ABB RAPID module: tester_left.mod

MODULE tester_left
LOCAL CONST string YuMi_App_Program_Version:="1.0.1"; !Do not edit or remove this line!
LOCAL VAR robtarget p35 := [[358.29,68.3,132.84],[0.2751,-0.0426083,0.86319,-0.421199],[-1,1,0,11],[117.327,9E+09,9E+09,9E+09,9E+09,9E+09]];
LOCAL VAR robtarget p34 := [[519.08,52.62,111.62],[0.0190745,-0.317014,0.947041,-0.0474542],[-2,1,-2,11],[179.331,9E+09,9E+09,9E+09,9E+09,9E+09]];
LOCAL VAR robtarget p33 := [[488.88,196.13,-9.51],[0.0436672,0.774832,-0.594672,-0.209984],[-2,0,-2,11],[-128.122,9E+09,9E+09,9E+09,9E+09,9E+09]];
LOCAL VAR robtarget p32 := [[438.93,-11.04,-14.27],[0.137086,0.640295,-0.744056,-0.132704],[-2,0,-2,11],[-135.659,9E+09,9E+09,9E+09,9E+09,9E+09]];
LOCAL VAR robtarget p31 := [[346.07,2.52,-21.9],[0.183409,0.628509,-0.722146,-0.223252],[-2,0,-2,11],[-129.96,9E+09,9E+09,9E+09,9E+09,9E+09]];
LOCAL VAR robtarget p30 := [[346.36,2.76,-22.07],[0.182499,0.628074,-0.72283,-0.223011],[-2,0,-2,11],[-129.954,9E+09,9E+09,9E+09,9E+09,9E+09]];
LOCAL VAR robtarget p29 := [[346.36,2.76,-22.07],[0.182498,0.628074,-0.722831,-0.22301],[-2,0,-2,11],[-129.954,9E+09,9E+09,9E+09,9E+09,9E+09]];
LOCAL VAR robtarget p28 := [[346.36,2.76,-22.07],[0.182497,0.628073,-0.722832,-0.223009],[-2,0,-2,11],[-129.954,9E+09,9E+09,9E+09,9E+09,9E+09]];
LOCAL VAR robtarget p27 := [[346.36,2.76,-22.07],[0.182493,0.628073,-0.722833,-0.22301],[-2,0,-2,11],[-129.954,9E+09,9E+09,9E+09,9E+09,9E+09]];
LOCAL VAR robtarget p26 := [[346.36,2.76,-22.07],[0.182492,0.628071,-0.722834,-0.223011],[-2,0,-2,11],[-129.954,9E+09,9E+09,9E+09,9E+09,9E+09]];
LOCAL VAR robtarget p25 := [[346.36,2.76,-22.07],[0.182489,0.628071,-0.722835,-0.22301],[-2,0,-2,11],[-129.954,9E+09,9E+09,9E+09,9E+09,9E+09]];
LOCAL VAR robtarget p24 := [[346.37,2.77,-22.07],[0.182481,0.628066,-0.722841,-0.223011],[-2,0,-2,11],[-129.954,9E+09,9E+09,9E+09,9E+09,9E+09]];
LOCAL VAR robtarget p23 := [[346.37,2.77,-22.08],[0.182475,0.628061,-0.722847,-0.22301],[-2,0,-2,11],[-129.954,9E+09,9E+09,9E+09,9E+09,9E+09]];
LOCAL VAR robtarget p22 := [[346.37,2.77,-22.08],[0.182471,0.628058,-0.722852,-0.223008],[-2,0,-2,11],[-129.954,9E+09,9E+09,9E+09,9E+09,9E+09]];
LOCAL VAR robtarget p21 := [[346.37,2.77,-22.08],[0.182457,0.628053,-0.72286,-0.223006],[-2,0,-2,11],[-129.954,9E+09,9E+09,9E+09,9E+09,9E+09]];
LOCAL VAR robtarget p20 := [[346.39,2.81,-22.09],[0.182382,0.628009,-0.722913,-0.223019],[-2,0,-2,11],[-129.952,9E+09,9E+09,9E+09,9E+09,9E+09]];
LOCAL VAR robtarget p19 := [[346.92,3.05,-22.39],[0.18104,0.627419,-0.724003,-0.222238],[-2,0,-2,11],[-129.95,9E+09,9E+09,9E+09,9E+09,9E+09]];
LOCAL VAR robtarget p18 := [[367.84,3.92,14.47],[0.223286,0.640903,-0.702206,-0.215161],[-2,0,-2,11],[-130.827,9E+09,9E+09,9E+09,9E+09,9E+09]];
LOCAL VAR robtarget p17 := [[412.3,51.52,46.99],[0.26981,0.654674,-0.703812,-0.0570357],[-2,0,-2,11],[-126.803,9E+09,9E+09,9E+09,9E+09,9E+09]];
LOCAL VAR robtarget p16 := [[496.94,50.54,-0.5],[0.0852698,-0.611194,0.718186,-0.321526],[-2,0,-1,1010],[-139.426,9E+09,9E+09,9E+09,9E+09,9E+09]];
LOCAL VAR robtarget p15 := [[500.11,217.09,68.79],[0.372259,-0.540285,0.603529,-0.453064],[-2,0,-1,1010],[-136.231,9E+09,9E+09,9E+09,9E+09,9E+09]];
LOCAL VAR robtarget p14 := [[409.25,103.49,24.74],[0.422813,-0.52314,0.597648,-0.436314],[-2,0,-1,1010],[-146.03,9E+09,9E+09,9E+09,9E+09,9E+09]];
LOCAL VAR robtarget p13 := [[321.14,2.68,-3.7],[0.326511,-0.570175,0.616333,-0.434079],[-2,0,-1,1010],[-149.503,9E+09,9E+09,9E+09,9E+09,9E+09]];
LOCAL VAR robtarget p12 := [[323.71,20.37,-12.88],[0.347699,-0.567053,0.614733,-0.423862],[-2,0,-1,1010],[-149.327,9E+09,9E+09,9E+09,9E+09,9E+09]];
LOCAL VAR robtarget p11 := [[318.83,3.47,-66.12],[0.377646,-0.544178,0.635778,-0.396283],[-2,0,-1,1010],[-148.179,9E+09,9E+09,9E+09,9E+09,9E+09]];
LOCAL VAR robtarget p10 := [[319.84,5.22,-58.84],[0.383222,-0.546134,0.616372,-0.418288],[-2,0,-1,1010],[-147.982,9E+09,9E+09,9E+09,9E+09,9E+09]];
LOCAL VAR robtarget p9 := [[328.17,3.84,-35.32],[0.291971,-0.584613,0.689413,-0.312553],[-2,0,-1,1010],[-148.669,9E+09,9E+09,9E+09,9E+09,9E+09]];
LOCAL VAR robtarget p8 := [[337.64,30.76,-7.64],[0.0603166,-0.700953,0.706625,-0.0755479],[-2,-1,-1,1010],[-140.725,9E+09,9E+09,9E+09,9E+09,9E+09]];
LOCAL VAR robtarget p7 := [[339.22,39.97,2.31],[0.254333,0.704549,-0.624556,-0.221031],[-2,-2,0,1010],[-142.847,9E+09,9E+09,9E+09,9E+09,9E+09]];
LOCAL VAR robtarget p6 := [[280.93,-22.19,-89.26],[0.280661,0.753652,-0.552241,-0.219698],[-2,-2,0,1010],[-144.058,9E+09,9E+09,9E+09,9E+09,9E+09]];
LOCAL VAR robtarget p5 := [[282.32,-20.83,-89.42],[0.275747,0.742915,-0.569862,-0.217482],[-2,-2,0,1010],[-144.216,9E+09,9E+09,9E+09,9E+09,9E+09]];
LOCAL VAR robtarget p4 := [[286.48,-20.76,-86.12],[0.126721,0.794038,-0.590704,-0.0671829],[-2,-1,-1,1010],[-143.981,9E+09,9E+09,9E+09,9E+09,9E+09]];
LOCAL VAR robtarget p3 := [[304.13,-11.5,-50.26],[0.0519145,0.826957,-0.559517,-0.0197134],[-2,-1,-1,1010],[-154.754,9E+09,9E+09,9E+09,9E+09,9E+09]];
LOCAL VAR robtarget p2 := [[316.65,45.52,21.47],[0.0502929,0.702983,-0.635561,0.315196],[-1,0,-1,1010],[-169.577,9E+09,9E+09,9E+09,9E+09,9E+09]];
LOCAL VAR robtarget p1 := [[358.29,68.3,132.84],[0.275101,-0.0426095,0.86319,-0.421198],[-1,1,0,11],[117.327,9E+09,9E+09,9E+09,9E+09,9E+09]];
LOCAL VAR robtarget s35 := [[358.29,68.3,132.84],[0.2751,-0.0426083,0.86319,-0.421199],[-1,1,0,11],[117.327,9E+09,9E+09,9E+09,9E+09,9E+09]];
LOCAL VAR robtarget s34 := [[519.08,52.62,111.62],[0.0190745,-0.317014,0.947041,-0.0474542],[-2,1,-2,11],[179.331,9E+09,9E+09,9E+09,9E+09,9E+09]];
LOCAL VAR robtarget s33 := [[488.88,196.13,-9.51],[0.0436672,0.774832,-0.594672,-0.209984],[-2,0,-2,11],[-128.122,9E+09,9E+09,9E+09,9E+09,9E+09]];
LOCAL VAR robtarget s32 := [[438.93,-11.04,-14.27],[0.137086,0.640295,-0.744056,-0.132704],[-2,0,-2,11],[-135.659,9E+09,9E+09,9E+09,9E+09,9E+09]];
LOCAL VAR robtarget s31 := [[346.07,2.52,-21.9],[0.183409,0.628509,-0.722146,-0.223252],[-2,0,-2,11],[-129.96,9E+09,9E+09,9E+09,9E+09,9E+09]];
LOCAL VAR robtarget s30 := [[346.36,2.76,-22.07],[0.182499,0.628074,-0.72283,-0.223011],[-2,0,-2,11],[-129.954,9E+09,9E+09,9E+09,9E+09,9E+09]];
LOCAL VAR robtarget s29 := [[346.36,2.76,-22.07],[0.182498,0.628074,-0.722831,-0.22301],[-2,0,-2,11],[-129.954,9E+09,9E+09,9E+09,9E+09,9E+09]];
LOCAL VAR robtarget s28 := [[346.36,2.76,-22.07],[0.182497,0.628073,-0.722832,-0.223009],[-2,0,-2,11],[-129.954,9E+09,9E+09,9E+09,9E+09,9E+09]];
LOCAL VAR robtarget s27 := [[346.36,2.76,-22.07],[0.182493,0.628073,-0.722833,-0.22301],[-2,0,-2,11],[-129.954,9E+09,9E+09,9E+09,9E+09,9E+09]];
LOCAL VAR robtarget s26 := [[346.36,2.76,-22.07],[0.182492,0.628071,-0.722834,-0.223011],[-2,0,-2,11],[-129.954,9E+09,9E+09,9E+09,9E+09,9E+09]];
LOCAL VAR robtarget s25 := [[346.36,2.76,-22.07],[0.182489,0.628071,-0.722835,-0.22301],[-2,0,-2,11],[-129.954,9E+09,9E+09,9E+09,9E+09,9E+09]];
LOCAL VAR robtarget s24 := [[346.37,2.77,-22.07],[0.182481,0.628066,-0.722841,-0.223011],[-2,0,-2,11],[-129.954,9E+09,9E+09,9E+09,9E+09,9E+09]];
LOCAL VAR robtarget s23 := [[346.37,2.77,-22.08],[0.182475,0.628061,-0.722847,-0.22301],[-2,0,-2,11],[-129.954,9E+09,9E+09,9E+09,9E+09,9E+09]];
LOCAL VAR robtarget s22 := [[346.37,2.77,-22.08],[0.182471,0.628058,-0.722852,-0.223008],[-2,0,-2,11],[-129.954,9E+09,9E+09,9E+09,9E+09,9E+09]];
LOCAL VAR robtarget s21 := [[346.37,2.77,-22.08],[0.182457,0.628053,-0.72286,-0.223006],[-2,0,-2,11],[-129.954,9E+09,9E+09,9E+09,9E+09,9E+09]];
LOCAL VAR robtarget s20 := [[346.39,2.81,-22.09],[0.182382,0.628009,-0.722913,-0.223019],[-2,0,-2,11],[-129.952,9E+09,9E+09,9E+09,9E+09,9E+09]];
LOCAL VAR robtarget s19 := [[346.92,3.05,-22.39],[0.18104,0.627419,-0.724003,-0.222238],[-2,0,-2,11],[-129.95,9E+09,9E+09,9E+09,9E+09,9E+09]];
LOCAL VAR robtarget s18 := [[367.84,3.92,14.47],[0.223286,0.640903,-0.702206,-0.215161],[-2,0,-2,11],[-130.827,9E+09,9E+09,9E+09,9E+09,9E+09]];
LOCAL VAR robtarget s17 := [[412.3,51.52,46.99],[0.26981,0.654674,-0.703812,-0.0570357],[-2,0,-2,11],[-126.803,9E+09,9E+09,9E+09,9E+09,9E+09]];
LOCAL VAR robtarget s16 := [[496.94,50.54,-0.5],[0.0852698,-0.611194,0.718186,-0.321526],[-2,0,-1,1010],[-139.426,9E+09,9E+09,9E+09,9E+09,9E+09]];
LOCAL VAR robtarget s15 := [[500.11,217.09,68.79],[0.372259,-0.540285,0.603529,-0.453064],[-2,0,-1,1010],[-136.231,9E+09,9E+09,9E+09,9E+09,9E+09]];
LOCAL VAR robtarget s14 := [[409.25,103.49,24.74],[0.422813,-0.52314,0.597648,-0.436314],[-2,0,-1,1010],[-146.03,9E+09,9E+09,9E+09,9E+09,9E+09]];
LOCAL VAR robtarget s13 := [[321.14,2.68,-3.7],[0.326511,-0.570175,0.616333,-0.434079],[-2,0,-1,1010],[-149.503,9E+09,9E+09,9E+09,9E+09,9E+09]];
LOCAL VAR robtarget s12 := [[323.71,20.37,-12.88],[0.347699,-0.567053,0.614733,-0.423862],[-2,0,-1,1010],[-149.327,9E+09,9E+09,9E+09,9E+09,9E+09]];
LOCAL VAR robtarget s11 := [[318.83,3.47,-66.12],[0.377646,-0.544178,0.635778,-0.396283],[-2,0,-1,1010],[-148.179,9E+09,9E+09,9E+09,9E+09,9E+09]];
LOCAL VAR robtarget s10 := [[319.84,5.22,-58.84],[0.383222,-0.546134,0.616372,-0.418288],[-2,0,-1,1010],[-147.982,9E+09,9E+09,9E+09,9E+09,9E+09]];
LOCAL VAR robtarget s9 := [[328.17,3.84,-35.32],[0.291971,-0.584613,0.689413,-0.312553],[-2,0,-1,1010],[-148.669,9E+09,9E+09,9E+09,9E+09,9E+09]];
LOCAL VAR robtarget s8 := [[337.64,30.76,-7.64],[0.0603166,-0.700953,0.706625,-0.0755479],[-2,-1,-1,1010],[-140.725,9E+09,9E+09,9E+09,9E+09,9E+09]];
LOCAL VAR robtarget s7 := [[339.22,39.97,2.31],[0.254333,0.704549,-0.624556,-0.221031],[-2,-2,0,1010],[-142.847,9E+09,9E+09,9E+09,9E+09,9E+09]];
LOCAL VAR robtarget s6 := [[280.93,-22.19,-89.26],[0.280661,0.753652,-0.552241,-0.219698],[-2,-2,0,1010],[-144.058,9E+09,9E+09,9E+09,9E+09,9E+09]];
LOCAL VAR robtarget s5 := [[282.32,-20.83,-89.42],[0.275747,0.742915,-0.569862,-0.217482],[-2,-2,0,1010],[-144.216,9E+09,9E+09,9E+09,9E+09,9E+09]];
LOCAL VAR robtarget s4 := [[286.48,-20.76,-86.12],[0.126721,0.794038,-0.590704,-0.0671829],[-2,-1,-1,1010],[-143.981,9E+09,9E+09,9E+09,9E+09,9E+09]];
LOCAL VAR robtarget s3 := [[304.13,-11.5,-50.26],[0.0519145,0.826957,-0.559517,-0.0197134],[-2,-1,-1,1010],[-154.754,9E+09,9E+09,9E+09,9E+09,9E+09]];
LOCAL VAR robtarget s2 := [[316.65,45.52,21.47],[0.0502929,0.702983,-0.635561,0.315196],[-1,0,-1,1010],[-169.577,9E+09,9E+09,9E+09,9E+09,9E+09]];
LOCAL VAR robtarget s1 := [[358.29,68.3,132.84],[0.275101,-0.0426095,0.86319,-0.421198],[-1,1,0,11],[117.327,9E+09,9E+09,9E+09,9E+09,9E+09]];
PROC main()
MoveSync s1;
OpenHand;
MoveSync s2;
MoveSync s3;
MoveSync s4;
MoveSync s5;
MoveSync s6;
CloseHand;
MoveSync s7;
MoveSync s8;
MoveSync s9;
MoveSync s10;
MoveSync s11;
OpenHand;
MoveSync s12;
MoveSync s13;
MoveSync s14;
MoveSync s15;
MoveSync s16;
MoveSync s17;
MoveSync s18;
MoveSync s19;
CloseHand;
MoveSync s20;
MoveSync s21;
MoveSync s22;
MoveSync s23;
MoveSync s24;
MoveSync s25;
MoveSync s26;
MoveSync s27;
MoveSync s28;
MoveSync s29;
MoveSync s30;
MoveSync s31;
OpenHand;
MoveSync s32;
MoveSync s33;
MoveSync s34;
MoveSync s35;
Move p1;
OpenHand;
Move p2;
Move p3;
Move p4;
Move p5;
Move p6;
CloseHand;
Move p7;
Move p8;
Move p9;
Move p10;
Move p11;
OpenHand;
Move p12;
Move p13;
Move p14;
Move p15;
Move p16;
Move p17;
Move p18;
Move p19;
CloseHand;
Move p20;
Move p21;
Move p22;
Move p23;
Move p24;
Move p25;
Move p26;
Move p27;
Move p28;
Move p29;
Move p30;
Move p31;
OpenHand;
Move p32;
Move p33;
Move p34;
Move p35;
ENDPROC
ENDMODULE
